Fanuc KAREL source: kf00107.KL

PROGRAM KF00107
%STACKSIZE=65535
%PRIORITY=65535
%NOLOCKGROUP
VAR
I : INTEGER
J : INTEGER
X : REAL
Y : REAL
B : BOOLEAN
C : BOOLEAN
TXT : STRING[80]
TXT2 : STRING[80]
AI : ARRAY[4] OF INTEGER
BI : ARRAY[4] OF INTEGER
P : XYZWPR
JP : JOINTPOS9
PF : POSITION
V1 : VECTOR
V2 : VECTOR
STATUS : INTEGER
BEGIN
I=1
X=1.0
B=TRUE
-- UNSAFE_SOURCE_IR line 24: B = native_io_value(1, 1)
END KF00107
